FUNCTION_BLOCK FB_MoveStepperAbs
VAR_INPUT
	stepsToMove				: INT;
	PosCurrent				: UDINT;
END_VAR
VAR_OUTPUT
END_VAR
VAR
	Step 					: INT := 0;
	bPowerOn				: INT;

END_VAR

MAIN.fbAxis1.bEnable := TRUE;

CASE Step OF
0:
	MAIN.fbAxis1.moveAbsPosition := 0.0;
	MAIN.fbAxis1.moveAbsVel := 0.0;
	MAIN.fbAxis1.bMoveAbsExe := FALSE;
	MAIN.fbAxis1.bHaltExe := FALSE;
	Step := 1;
1:

	IF MAIN.fbAxis1.bPwrStatus THEN
		MAIN.fbAxis1.moveAbsPosition := stepsToMove;
		MAIN.fbAxis1.moveAbsVel := 100;
		MAIN.fbAxis1.bMoveAbsExe := TRUE;
		IF MAIN.fbAxis1.bMoveAbsDone THEN
			MAIN.fbAxis1.bMoveAbsExe := FALSE;
			MAIN.fbAxis1.bHaltExe := TRUE;
			Step := 2;
		END_IF
	END_IF	
2:
	IF MAIN.fbAxis1.bHaltDone = TRUE THEN
		MAIN.fbAxis1.bHaltExe := FALSE;
	END_IF

	MAIN.bMoveAbsolute := FALSE;
	
	Step := 0;
END_CASE

END_FUNCTION_BLOCK

(* stored: Version 1.1.0.1, ProductVersion 3.1.4024.9
   POU FB_MoveStepperAbs: Id {9fd65aaa-dbc3-43b1-8b0c-e64e3a5d47b1}, SpecialFunc None *)
